Fanuc KAREL source: kb00148.KL

-- PROVISIONAL review KL for V1013-1; original PC SHA256 0778a1f18c290424ee859c154a3295477165c5f5d6ecfc277ff83830c8f35da3
-- Incomplete behavior may be omitted. Consult companion uncertainty JSON. Do not deploy.
PROGRAM KB00148
%NOLOCKGROUP
BEGIN
  -- UNRESOLVED_PC offsets 5-14; opcodes 3F,75
  -- UNRESOLVED_PC offsets 19-28; opcodes 3F,75
  -- UNRESOLVED_PC offsets 33-40; opcodes 9D,23
  -- UNRESOLVED_PC offsets 45-71; opcodes 27,22,2A,22,2A,22,31
  -- UNRESOLVED_PC offsets 76-80; opcodes 7F
END KB00148
